(*!
<summary>Places the cursor before the first source entry.</summary>
<description>
The next MoveNext starts at zero. Does not modify the source or release payload; reading Current now yields an
empty descriptor. Descendants cannot override this cursor operation; advancement, reset and borrowed current
views use the same cursor state.
</description>
*)
{attribute "object_name" := "Reset"}
METHOD FINAL Reset
_CurrentIndex := -1;
END_METHOD

(*!
<summary>Reports the size of this function-block instance.</summary>
<description>
Measured in bytes; includes inline storage but excludes separately allocated buffers, payload and enumerators.
</description>
*)
{attribute 'monitoring' := 'call'}
PROPERTY SelfSize : ULINT
GET
SelfSize := XSIZEOF(THIS^);
END_GET
END_PROPERTY

(*!
<summary>Requires the configured source before traversal or current-value access.</summary>
<description>
A missing mandatory source is configuration failure, not an empty collection. Raises a framework diagnostic
outside lifecycle methods and before mutation; it does not validate arbitrary pointer lifetime.
</description>
*)
METHOD PRIVATE requireSource
IF _Queue = 0 THEN
	TOF_Core.Exceptions.ThrowDataMemberNotSpecified(
		sourceNamespaceName := NamespaceName,
		sourceClassName := ClassName,
		sourcePOUName := __POUNAME(),
		sourcePosition := __POSITION(),
		dataMemberName := 'queue'
	);
END_IF
END_METHOD

END_FUNCTION_BLOCK

// ---- Stack/Stack.TcPOU
(*
SPDX-FileCopyrightText: © 2026 Oleksandr Tiutyk <trofimich@gmail.com>
SPDX-License-Identifier: MIT
License: https://opensource.org/license/mit
*)

(*!
<summary>Stores generic values for last-in, first-out processing.</summary>
<description>
CreateEnumerator allocates an independent cursor owned by its caller. The collection must remain alive while
that cursor is used. Successful insertion transfers disposal responsibility for owned payload; borrowed
payload must remain alive while stored. The caller-side descriptor copy is not reset and must not be released
again after transfer. Independent owning aliases and overlapping owned allocations are unsupported. Peek and
GetByIndex borrow entries. RemoveLast releases the top without shifting remaining entries. Indices and
enumeration run from top to bottom. Static capacity defaults to ten; zero selects dynamic storage. Validators
are borrowed for the collection lifetime. ContainsGeneric defaults to releasing its query. Growth checks
allocation arithmetic and invokes the terminal mechanism on null NEW before replacing the old buffer. No
locking or mutation-version checks are implemented. Generic lookup with requested query release also attempts
cleanup on lookup failure before propagating the captured exception; terminal OOM takes precedence.
Instances cannot be assigned by value: copying backing pointers or disposal responsibility would create
unsafe aliases. Interface references still borrow this instance; copying an interface does not clone storage.
</description>
*)

{attribute 'no_explicit_call' := 'do not call this function block directly'}
FUNCTION_BLOCK FINAL Stack 
VAR_GENERIC CONSTANT
	//!<summary>Inline descriptor capacity; zero selects dynamic backing storage.</summary>
	{attribute 'hide'} 
	_StaticCapacity : TOF_Core.DINT_LENGTH := 10;
END_VAR
EXTENDS TOF_Core.Object IMPLEMENTS IStack
VAR_INPUT
	//! <summary>Number of slots added when dynamic storage is full; must be positive when growth is required.</summary>
	DefaultDynamicAllocationElementCount : BYTE := 10;	
END_VAR
VAR_STAT
	//! <summary>Class name shared by all instances of this function block.</summary>
	{attribute 'hide'} 
	_ClassName : STRING := __POUNAME();
END_VAR
VAR	
	{attribute 'hide'} 
	_ValueValidator : TOF_Core.IGenericValueValidator;

	{attribute 'hide'} 
	_Array : POINTER TO TOF_Core.GENERIC_VALUE;
	{attribute 'hide'} 
	_StaticArray : ARRAY [0.._StaticCapacity - 1] OF TOF_Core.GENERIC_VALUE;
	
	{attribute 'hide'} 
	_DynamicCapacity : TOF_Core.DINT_LENGTH;
	{attribute 'hide'} 
	_Length : TOF_Core.DINT_LENGTH;
END_VAR

(*!
<summary>Expands the dynamic descriptor buffer.</summary>
<description>
Static instances return without allocation. A positive increment must fit DINT capacity and the UDINT
allocation-byte limit; invalid ranges raise ArgumentOutOfRangeException before storage changes. A null
allocation invokes the terminal allocation-failure mechanism before copying or deleting the old buffer.
Existing descriptors are moved without cloning payload; incoming ownership is not accepted by this helper.
</description>
*)
METHOD PROTECTED FINAL AllocateMemory 
VAR_INPUT
	elementCount : TOF_Core.DINT_LENGTH;
END_VAR
VAR CONSTANT
	//!<summary>Bytes per descriptor slot used to bound and size the dynamic backing allocation.</summary>
	ENTRY_ALLOCATION_SIZE : ULINT := XSIZEOF(TOF_Core.GENERIC_VALUE);
END_VAR
VAR
	newMemory : POINTER TO TOF_Core.GENERIC_VALUE;
	newCapacity : ULINT;

END_VAR
IF NOT Dynamic THEN
	RETURN;
END_IF

IF elementCount <= TOF_Core.SignedInt32.ZERO THEN
	TOF_Core.Exceptions.ThrowArgumentOutOfRange(
		sourceNamespaceName := NamespaceName,
		sourceClassName := ClassName,
		sourcePOUName := __POUNAME(),
		sourcePosition := __POSITION(),
		argumentName := 'elementCount',
		argumentValue := elementCount
	);
END_IF

newCapacity := TO_ULINT(_DynamicCapacity) + TO_ULINT(elementCount);

IF newCapacity > TO_ULINT(TOF_Core.SignedInt32.MAX_VALUE)
	OR_ELSE newCapacity > TO_ULINT(TOF_Core.UnsignedInt32.MAX_VALUE) / ENTRY_ALLOCATION_SIZE
THEN
	TOF_Core.Exceptions.ThrowArgumentOutOfRange(
		sourceNamespaceName := NamespaceName,
		sourceClassName := ClassName,
		sourcePOUName := __POUNAME(),
		sourcePosition := __POSITION(),
		argumentName := 'capacity',
		argumentValue := newCapacity
	);
END_IF

newMemory := __NEW(BYTE, TO_UDINT(ENTRY_ALLOCATION_SIZE * newCapacity));

IF newMemory = 0 THEN
	TOF_Core.DynamicMemoryManager.RaiseAllocationFailure();
END_IF

IF _Length > TOF_Core.SignedInt32.ZERO THEN
	Tc2_System.MEMCPY(destAddr := newMemory, srcAddr := _Array, n := TO_UDINT(ENTRY_ALLOCATION_SIZE * TO_ULINT(_Length)));
END_IF

IF _Array <> 0 THEN
	__DELETE(_Array);
END_IF

_DynamicCapacity := TO_DINT(newCapacity);
_Array := newMemory;
END_METHOD

(*!
<summary>Reports the currently allocated number of slots.</summary>
<description>
Units are stack entries. Static capacity is fixed; dynamic capacity can change on growth or clearing. This is
not a guarantee that the next allocation succeeds.
</description>
*)
{attribute 'monitoring' := 'call'}
PROPERTY FINAL Capacity : TOF_Core.DINT_LENGTH
GET
Capacity := SEL(_StaticCapacity = TOF_Core.SignedInt32.ZERO, _StaticCapacity, _DynamicCapacity);
END_GET
END_PROPERTY

(*!
<summary>Borrows the concrete collection class name without transferring storage ownership.</summary>
*)
{attribute 'monitoring' := 'call'}
PROPERTY ClassName : REFERENCE TO STRING
GET
ClassName REF= _ClassName;
END_GET
END_PROPERTY

(*!
<summary>Removes all entries and releases dynamic backing storage.</summary>
<description>
Owned payload is released best effort through GENERIC_VALUE.Release; borrowed storage is not freed. Static
capacity and the borrowed validator are retained. Dynamic capacity becomes zero. Returns this collection and
invalidates positions and views. Cleanup callbacks must not reenter mutation.
</description>
*)
METHOD Clear : IStack
VAR
	i : DINT;
END_VAR
Clear := THIS^;

FOR i := 0 TO _Length - 1 DO
	_Array[i].Release();
END_FOR

_Length := 0;
_DynamicCapacity := 0;

IF _Array <> 0 AND_THEN Dynamic THEN
	__DELETE(_Array);	
END_IF
END_METHOD

(*!
<summary>Searches for a value using default generic equality.</summary>
<description>
Borrows the ANY argument during a linear search without cloning or releasing it. isObject = TRUE means a live
Object FB instance, not a pointer or interface variable. Equality exceptions propagate; callbacks that mutate
the collection can invalidate traversal.
</description>
*)
METHOD Contains : BOOL
VAR_INPUT
	value : ANY;
	isObject : BOOL := FALSE;
END_VAR
VAR
	genericValue : TOF_Core.GENERIC_VALUE;
	i : TOF_Core.DINT_INDEX;
END_VAR

genericValue := TOF_Core.GenericValueFactory.FromAnyType(
		value := value,
		isObject := isObject,
		memoryManagementBehavior := TOF_Core.GENERIC_MEMORY_MANAGEMENT_BEHAVIOR.STORE_ORIGINAL_REFERENCE_AND_NOT_OWNS_MEMORY
	);

FOR i := 0 TO _Length - 1 DO
	IF _Array[i].Equals(otherValue := genericValue) THEN
		Contains := TRUE;
		RETURN;
	END_IF
END_FOR
END_METHOD

(*!
<summary>Searches for an equal generic value and optionally releases the query.</summary>
<description>
Uses GENERIC_VALUE.Equals in a linear search. releaseValue defaults to TRUE: after a completed search, Release
is called on the local query copy, including on a miss. Caller-side aliases are not reset. The query must not
own storage retained by the collection. Requested release is attempted after both successful lookup and lookup
failure. Before cleanup, the original framework exception is retained and a borrowed static system exception
is cloned to preserve its code, catch point and timestamps across cleanup callbacks. The captured exception is
then propagated through ExceptionManager.Throw in the current cyclic task; native errors use the framework
SystemException representation. If capturing the system exception fails with terminal OOM, query cleanup is
still attempted and terminal OOM takes precedence. Terminal allocation state is never cleared. Release is best
effort and does not prove successful deallocation. Cleanup callbacks must not reenter collection mutation.
</description>
*)
METHOD ContainsGeneric : BOOL
VAR_INPUT
	value : TOF_Core.GENERIC_VALUE;
	releaseValue : BOOL := TRUE;
END_VAR
VAR
	exceptionCode : __SYSTEM.ExceptionCode;
	caughtException : TOF_Core.IException;

	i : DINT;
END_VAR
__TRY
	FOR i := 0 TO _Length - 1 DO
		IF _Array[i].Equals(otherValue := value) THEN
			ContainsGeneric := TRUE;
			EXIT;
		END_IF
	END_FOR
__CATCH(exceptionCode)
	caughtException := TOF_Core.ExceptionManager.GetLastException(
		exceptionCode := exceptionCode,
		catchPointNamespaceName := NamespaceName,
		catchPointPOUName := __POUNAME(),
		catchPointPosition := __POSITION()
	);
__ENDTRY

IF releaseValue THEN
	IF caughtException <> 0 AND_THEN NOT caughtException.IsDynamicInstance THEN
		__TRY
			TOF_Core.DynamicMemoryManager.RaiseIfAllocationFailed();
			__QUERYINTERFACE(caughtException.Clone(), caughtException);
		__CATCH(exceptionCode)
			value.Release();

			TOF_Core.ExceptionManager.ReThrowLastException(
				exceptionCode := exceptionCode,
				catchPointNamespaceName := NamespaceName,
				catchPointPOUName := __POUNAME(),
				catchPointPosition := __POSITION()
			);
		__ENDTRY
	END_IF

	value.Release();
END_IF

IF caughtException <> 0 THEN
	TOF_Core.ExceptionManager.Throw(exception := caughtException);
END_IF
END_METHOD

(*!
<summary>Creates an independent enumerator owned by the caller.</summary>
<description>
The caller must explicitly release the enumerator and keep this collection alive while using it. Allocation
failure invokes DynamicMemoryManager.RaiseAllocationFailure without a heap exception; it is terminal and is
not returned as a recoverable null result.
</description>
*)
METHOD CreateEnumerator : TOF_Core.IEnumerator
VAR
	enumerator : POINTER TO StackEnumerator;
END_VAR
enumerator := __NEW(StackEnumerator(stack := THIS^));

IF enumerator = 0 THEN
	TOF_Core.DynamicMemoryManager.RaiseAllocationFailure();
END_IF

CreateEnumerator := enumerator^;
END_METHOD

(*!
<summary>Reports whether storage can grow dynamically.</summary>
<description>
Static capacity zero selects dynamic storage. Dynamic collections can still fail to allocate.
</description>
*)
{attribute 'monitoring' := 'call'}
PROPERTY FINAL Dynamic : BOOL
GET
Dynamic := _StaticCapacity = TOF_Core.SignedInt32.ZERO;
END_GET
END_PROPERTY

(*!
<summary>Reports whether the collection has no entries.</summary>
<description>
Reflects Length; not a check of payload lifetime or memory health.
</description>
*)
{attribute 'monitoring' := 'call'}
PROPERTY FINAL Empty : BOOL
GET
Empty := _Length <= TOF_Core.SignedInt32.ZERO;
END_GET
END_PROPERTY

(*!
<summary>Releases owned payload and backing storage during destruction.</summary>
<description>
Calls Clear; lifecycle methods and payload cleanup callbacks must not raise exceptions or reenter mutation.
Payload release is best effort, not proof of successful destruction. No separate copy-code ownership handoff
is implemented.
</description>
*)

METHOD FB_exit : BOOL
VAR_INPUT
	bInCopyCode : BOOL; 
END_VAR
Clear();
END_METHOD

(*!
<summary>Binds the optional validator and inline storage during initialization.</summary>
<description>
The validator is borrowed and must remain alive while used; it is not invoked here. Static storage is bound
without allocation. Lifecycle methods must not raise exceptions. No explicit online-change relocation repair
is implemented.
</description>
*)
METHOD FB_init : BOOL
VAR_INPUT
	bInitRetains : BOOL; // TRUE: the retain variables are initialized (reset warm / reset cold)
	bInCopyCode : BOOL; // TRUE: the instance will be copied to the copy code afterward (online change)
	valueValidator : TOF_Core.IGenericValueValidator;
END_VAR
_ValueValidator := valueValidator;

IF NOT Dynamic THEN
	_Array := ADR(_StaticArray); 
END_IF
END_METHOD

(*!
<summary>Reports whether fixed-capacity storage has no free slot.</summary>
<description>
Dynamic collections report FALSE even when Length equals Capacity. This does not guarantee available heap
memory.
</description>
*)
{attribute 'monitoring' := 'call'}
PROPERTY FINAL Full : BOOL
GET
Full := _StaticCapacity <> TOF_Core.SignedInt32.ZERO AND_THEN _Length >= _StaticCapacity;
END_GET
END_PROPERTY

(*!
<summary>Borrows the descriptor at a zero-based stack position.</summary>
<description>
Position zero is the top; increasing indices move toward the bottom. An out-of-range index raises an
exception. Returned descriptors and payload are borrowed, not clones. Do not modify descriptor metadata or
release payload through this view, even when IsMemoryOwner is TRUE. Keep the source and borrowed storage
alive; mutation or destruction can invalidate the view.
</description>
*)
METHOD GetByIndex : REFERENCE TO TOF_Core.GENERIC_VALUE
VAR_INPUT
	index : TOF_Core.DINT_INDEX;
END_VAR
IF index < TOF_Core.SignedInt32.ZERO OR_ELSE index >= _Length THEN
	TOF_Core.Exceptions.ThrowArgumentOutOfRange(
		sourceNamespaceName := NamespaceName,
		sourceClassName := ClassName,
		sourcePOUName := __POUNAME(),
		sourcePosition := __POSITION(),
		argumentName := 'index',
		argumentValue := index
	);
END_IF

GetByIndex REF= _Array[_Length - 1 - index];
END_METHOD

(*!
<summary>Reports the number of stored entries.</summary>
<description>
Units are stack entries. Existing positions range from zero through Length minus one.
</description>
*)
{attribute 'monitoring' := 'call'}
PROPERTY FINAL Length : TOF_Core.DINT_LENGTH
GET
Length := _Length;
END_GET
END_PROPERTY

(*!
<summary>Provides the library namespace for diagnostics.</summary>
<description>
Borrowed read-only reference to compiler-initialized metadata; no ownership transfer.
</description>
*)
{attribute 'monitoring' := 'call'}
PROPERTY NamespaceName : REFERENCE TO STRING
GET
NamespaceName REF= CurrentNamespace.Name;
END_GET
END_PROPERTY

(*!
<summary>Borrows the LIFO top without removing it.</summary>
<description>
An empty stack raises CollectionEmptyException. Returned descriptors and payload are borrowed, not clones. Do
not modify descriptor metadata or release payload through this view, even when IsMemoryOwner is TRUE. Keep the
source and borrowed storage alive; mutation or destruction can invalidate the view.
</description>
*)
METHOD Peek : REFERENCE TO TOF_Core.GENERIC_VALUE
IF _Length <= TOF_Core.SignedInt32.ZERO THEN
	TOF_Core.Exceptions.ThrowCollectionEmpty(
		sourceNamespaceName := NamespaceName,
		sourceClassName := ClassName,
		sourcePOUName := __POUNAME(),
		sourcePosition := __POSITION(),
		collectionName := GetName()
	);
END_IF

Peek REF= _Array[_Length - 1];
END_METHOD

(*!
<summary>Copies a value and appends it to the stack top.</summary>
<description>
Borrows the original during the call. isObject = TRUE requires a live Object FB instance implementing
ICloneable; other data is copied as bytes without recursively cloning references. A prepared copy is released
if insertion fails before acceptance; exceptions propagate. Engine-managed exception objects are unsupported.
The original failure is captured before cleanup so nested cleanup handling cannot replace its payload.
A static native wrapper is cloned before cleanup; failure to capture still attempts prepared-copy disposal.
Terminal allocation failure takes precedence and no exception clone is allocated after its latch is set.
</description>
*)
METHOD PushCopy : IStack
VAR_INPUT
	value : ANY;
	isObject : BOOL := FALSE;
END_VAR
VAR
	exceptionCode : __SYSTEM.ExceptionCode;
	caughtException : TOF_Core.IException;
	genericValue : TOF_Core.GENERIC_VALUE;
END_VAR

genericValue := TOF_Core.GenericValueFactory.FromAnyType(
		value := value,
		isObject := isObject,
		memoryManagementBehavior := TOF_Core.GENERIC_MEMORY_MANAGEMENT_BEHAVIOR.CLONE_ORIGINAL_VALUE_AND_OWNS_MEMORY
	);

__TRY
	PushCopy := PushGeneric(value := genericValue);
__CATCH(exceptionCode)
	caughtException := TOF_Core.ExceptionManager.GetLastException(
		exceptionCode := exceptionCode,
		catchPointNamespaceName := NamespaceName,
		catchPointPOUName := __POUNAME(),
		catchPointPosition := __POSITION()
	);
__ENDTRY

IF caughtException <> 0 THEN
	__TRY
		TOF_Core.DynamicMemoryManager.RaiseIfAllocationFailed();

		IF NOT caughtException.IsDynamicInstance THEN
			__QUERYINTERFACE(caughtException.Clone(), caughtException);
		END_IF
	__CATCH(exceptionCode)
		genericValue.Release();

		TOF_Core.ExceptionManager.ReThrowLastException(
			exceptionCode := exceptionCode,
			catchPointNamespaceName := NamespaceName,
			catchPointPOUName := __POUNAME(),
			catchPointPosition := __POSITION()
		);
	__ENDTRY

	genericValue.Release();

	TOF_Core.ExceptionManager.Throw(exception := caughtException);
END_IF
END_METHOD

(*!
<summary>Pushes a descriptor onto the stack top.</summary>
<description>
Successful insertion transfers disposal responsibility for owned payload; borrowed payload must remain alive
while stored. The caller-side descriptor copy is not reset and must not be released again after transfer.
Independent owning aliases and overlapping owned allocations are unsupported. Full static storage raises an
exception. A configured validator is invoked once before any capacity growth or ownership acceptance.
Validation failure leaves the buffer, Length and incoming ownership unchanged; its exception propagates.
Validator callbacks must not mutate this collection.
</description>
*)
METHOD PushGeneric : IStack
VAR_INPUT
	value : TOF_Core.GENERIC_VALUE;
END_VAR
IF _ValueValidator <> 0 THEN
	_ValueValidator.Validate(validatedObjectName := GetName(), valueToValidate := value);
END_IF

IF _Length >= Capacity THEN
	IF Dynamic THEN
		AllocateMemory(elementCount := DefaultDynamicAllocationElementCount);
	ELSE
		TOF_Core.Exceptions.ThrowStaticCollectionFull(
			sourceNamespaceName := NamespaceName,
			sourceClassName := ClassName,
			sourcePOUName := __POUNAME(),
			sourcePosition := __POSITION(),
			collectionName := GetName(),
			capacity := TO_UDINT(Capacity)
		);
	END_IF
END_IF

PushGeneric := THIS^;

_Array[_Length] := value;
_Length := _Length + 1;
END_METHOD

(*!
<summary>Removes and releases the LIFO top.</summary>
<description>
An empty stack raises CollectionEmptyException. Owned top storage is released best effort, not returned to the
caller. Remaining descriptors are not moved; removal takes constant time apart from payload cleanup. Returns
this stack; positions and views may change. Cleanup callbacks must not reenter mutation.
</description>
*)
METHOD RemoveLast : IStack
IF _Length <= TOF_Core.SignedInt32.ZERO THEN
	TOF_Core.Exceptions.ThrowCollectionEmpty(
		sourceNamespaceName := NamespaceName,
		sourceClassName := ClassName,
		sourcePOUName := __POUNAME(),
		sourcePosition := __POSITION(),
		collectionName := GetName()
	);
END_IF

_Length := _Length - 1;
_Array[_Length].Release();

RemoveLast := THIS^;
END_METHOD

(*!
<summary>Reports the size of this function-block instance.</summary>
<description>
Measured in bytes; includes inline storage but excludes separately allocated buffers, payload and enumerators.
</description>
*)
{attribute 'monitoring' := 'call'}
PROPERTY SelfSize : ULINT
GET
SelfSize := XSIZEOF(THIS^);
END_GET
END_PROPERTY

(*!
<summary>Exposes the configured value validator.</summary>
<description>
Borrowed optional reference fixed at initialization. Zero means no validator. The collection does not own or
release it.
</description>
*)
{attribute 'monitoring' := 'call'}
PROPERTY FINAL ValueValidator : TOF_Core.IGenericValueValidator
GET
ValueValidator := _ValueValidator;
END_GET
END_PROPERTY

END_FUNCTION_BLOCK

// ---- Stack/StackEnumerator.TcPOU
(*
SPDX-FileCopyrightText: © 2026 Oleksandr Tiutyk <trofimich@gmail.com>
SPDX-License-Identifier: MIT
License: https://opensource.org/license/mit
*)

(*!
<summary>Enumerates a borrowed stack using an independent cursor.</summary>
<description>
The source must be non-null, outlive the cursor and remain structurally unchanged during traversal. The caller
explicitly releases a dynamically created cursor. Current is borrowed read-only data, never an ownership
transfer. Traverses from top to bottom. Supports both fixed-capacity and dynamic stacks. MoveNext stops
advancing at the end position of an unchanged source; repeated exhausted calls return FALSE until Reset.
A null constructor source is diagnosed by traversal/current access, never by FB_init.
</description>
*)

{attribute 'no_explicit_call' := 'do not call this function block directly'}
{attribute 'enable_dynamic_creation'}
FUNCTION_BLOCK StackEnumerator EXTENDS TOF_Core.Object IMPLEMENTS TOF_Core.IEnumerator
VAR_STAT
	//! <summary>Class name shared by all instances of this function block.</summary>
	{attribute 'hide'} 
	_ClassName : STRING := __POUNAME();
END_VAR
VAR
	{attribute 'hide'} 
	_Stack : IReadOnlyStack;
	{attribute 'hide'} 
	//!<summary>Top-relative position; minus one represents the cursor before the first entry.</summary>
	_CurrentIndex : DINT := -1;
	
	{attribute 'hide'} 
	_GenericValue : TOF_Core.GENERIC_VALUE;
END_VAR

(*!
<summary>Borrows the concrete cursor class name without transferring storage ownership.</summary>
*)
{attribute 'monitoring' := 'call'}
PROPERTY ClassName : REFERENCE TO STRING
GET
ClassName REF= _ClassName;
END_GET
END_PROPERTY

(*!
<summary>Exposes a read-only borrowed view of the current entry.</summary>
<description>
Reading Current before the first successful MoveNext, after Reset or after exhaustion yields an empty
descriptor. Otherwise payload is borrowed, with no disposal rights. Do not modify or release the descriptor.
The view may change on subsequent property access, cursor movement or source mutation.
Missing source raises DataMemberNotSpecifiedException before source access or cursor advancement.
</description>
*)
{attribute 'monitoring' := 'call'}
PROPERTY FINAL Current : REFERENCE TO TOF_Core.GENERIC_VALUE
GET
requireSource();

IF _CurrentIndex >= TOF_Core.SignedInt32.ZERO AND_THEN _CurrentIndex < _Stack.Length THEN
	_GenericValue := _Stack.GetByIndex(index := _CurrentIndex); 
ELSE
	_GenericValue.Reset();	
END_IF 

Current REF= _GenericValue;
END_GET
END_PROPERTY

(*!
<summary>Binds the borrowed source for enumeration.</summary>
<description>
The source must be non-null and outlive the cursor. Only the reference is assigned; no allocation, callbacks
or throwing validation are performed. A null source remains invalid configuration and is reported by
MoveNext or current-value access without throwing from initialization.
</description>
*)
METHOD FB_init : BOOL
VAR_INPUT
	bInitRetains : BOOL; // TRUE: the retain variables are initialized (reset warm / reset cold)
	bInCopyCode : BOOL;  // TRUE: the instance will be copied to the copy code afterward (online change)
	stack : IReadOnlyStack;
END_VAR
_Stack := stack;
END_METHOD

(*!
<summary>Advances the cursor to the next source position.</summary>
<description>
The source must be live, non-null and structurally unchanged during traversal. TRUE identifies a current
entry. The index advances only while below source Length and stops at the end position. Repeated exhausted
calls return FALSE without incrementing the index; reading Current yields an empty descriptor. Reset allows
traversal from the beginning again. No snapshot or mutation detection is provided. Descendants cannot override
this cursor operation; advancement, reset and borrowed current views use the same cursor state.
Missing source raises DataMemberNotSpecifiedException before source access or cursor advancement.
</description>
*)
{attribute "object_name" := "MoveNext"}
METHOD FINAL MoveNext : BOOL
requireSource();

IF _CurrentIndex < _Stack.Length THEN
	_CurrentIndex := _CurrentIndex + 1;
END_IF

MoveNext := _CurrentIndex < _Stack.Length;
END_METHOD

(*!
<summary>Provides the library namespace for diagnostics.</summary>
<description>
Borrowed read-only reference to compiler-initialized metadata; no ownership transfer.
</description>
*)
{attribute 'monitoring' := 'call'}
PROPERTY NamespaceName : REFERENCE TO STRING
GET
NamespaceName REF= CurrentNamespace.Name;
END_GET
END_PROPERTY

(*!
<summary>Places the cursor before the first source entry.</summary>
<description>
The next MoveNext starts at zero. Does not modify the source or release payload; reading Current now yields an
empty descriptor. Descendants cannot override this cursor operation; advancement, reset and borrowed current
views use the same cursor state.
</description>
*)
{attribute "object_name" := "Reset"}
METHOD FINAL Reset
_CurrentIndex := -1;
END_METHOD

(*!
<summary>Reports the size of this function-block instance.</summary>
<description>
Measured in bytes; includes inline storage but excludes separately allocated buffers, payload and enumerators.
</description>
*)
{attribute 'monitoring' := 'call'}
PROPERTY SelfSize : ULINT
GET
SelfSize := XSIZEOF(THIS^);
END_GET
END_PROPERTY

(*!
<summary>Requires the configured source before traversal or current-value access.</summary>
<description>
A missing mandatory source is configuration failure, not an empty collection. Raises a framework diagnostic
outside lifecycle methods and before mutation; it does not validate arbitrary pointer lifetime.
</description>
*)
METHOD PRIVATE requireSource
IF _Stack = 0 THEN
	TOF_Core.Exceptions.ThrowDataMemberNotSpecified(
		sourceNamespaceName := NamespaceName,
		sourceClassName := ClassName,
		sourcePOUName := __POUNAME(),
		sourcePosition := __POSITION(),
		dataMemberName := 'stack'
	);
END_IF
END_METHOD

END_FUNCTION_BLOCK

// ---- UniqueDataSet/UniqueDataSet.TcPOU
(*
SPDX-FileCopyrightText: © 2026 Oleksandr Tiutyk <trofimich@gmail.com>
SPDX-License-Identifier: MIT
License: https://opensource.org/license/mit
*)

(*!
<summary>Stores unique generic values with fixed or dynamic capacity.</summary>
<description>
CreateEnumerator allocates an independent cursor owned by its caller. The collection must remain alive while
that cursor is used. SetGeneric replaces a matching entry with the incoming descriptor. SetGeneric preserves
disposal responsibility when the same allocation is reused; transferred caller-side owning aliases must not be
released again. Lookup uses GENERIC_VALUE equality/hashing or the borrowed valueEqualityComparer supplied once
through FB_init. Pass zero explicitly to use default value equality and hashing. Empty values are supported
unless rejected by a validator. Raw queries create borrowed descriptors with an explicit object flag. Entries
and enumeration have no guaranteed order; positions are storage slots, not sorted ranks. Do not modify stored
descriptors through returned references. Try lookup/removal operations contain exceptions without rolling back
partial effects. Generic query arguments are borrowed by default. Explicitly requested release in Try
operations is attempted even after lookup failure; caller-side owning aliases are not reset. Borrowed
elements, including OBJECT instances, remain caller-owned and must stay alive while stored. Do not delete
owned payload through external aliases. Keep equality/hash-relevant data and comparer configuration stable:
remove before changing them, then insert again. Fields unrelated to active equality/hash may change. Callbacks
must not mutate elements or reenter collection mutation; explicit query release must not dispose of retained
storage. Default OBJECT equality/hashing uses Object.Equals/GetHashCode; Clone has its own identity. Discard
and populate the index again after equality-relevant address relocation before further lookup. Static index
storage adds 12 bytes per capacity slot and three pointers plus the comparer reference. Dynamic entries and
the 12-byte-per-slot index share one allocation; growth temporarily retains both old and new allocations.
Expected bucket lookup is constant time plus hashing/equality costs, worst case linear; compaction and
rebuilding after removal are linear in capacity and Length. The validator is borrowed for the collection
lifetime. No internal locking is implemented. Concurrent access involving mutation requires caller
coordination; this implementation does not provide a concurrent-container guarantee. Generic lookup with
requested query release also attempts cleanup on lookup failure before propagating the captured exception;
terminal OOM takes precedence.
Instances cannot be assigned by value: copying backing pointers or disposal responsibility would create
unsafe aliases. Interface references still borrow this instance; copying an interface does not clone storage.
</description>
*)

{attribute 'no_explicit_call' := 'do not call this function block directly'}
FUNCTION_BLOCK UniqueDataSet
VAR_GENERIC CONSTANT
	{attribute 'hide'}
	//! <summary>Inline capacity; zero selects dynamic backing storage.</summary>
	_StaticCapacity : TOF_Core.DINT_LENGTH := 0;
END_VAR
EXTENDS TOF_Core.Object IMPLEMENTS IUniqueDataSet
VAR_INPUT
	//! <summary>Number of slots added when dynamic storage is full; must be positive when growth is required.</summary>
	DefaultDynamicAllocationElementCount : BYTE := 10;
END_VAR
VAR_STAT
	//! <summary>Class name shared by all instances of this function block.</summary>
	{attribute 'hide'}
	_ClassName : STRING := __POUNAME();
END_VAR
VAR
	{attribute 'hide'}
	_ValueValidator : TOF_Core.IGenericValueValidator;
	{attribute 'hide'}
	_ValueEqualityComparer : TOF_Core.IEqualityComparer;

	{attribute 'hide'}
	_Array : POINTER TO TOF_Core.GENERIC_VALUE;
	{attribute 'hide'}
	_StaticArray : ARRAY [0.._StaticCapacity - 1] OF TOF_Core.GENERIC_VALUE;

	{attribute 'hide'}
	_Hashes : POINTER TO UDINT;
	{attribute 'hide'}
	_Buckets : POINTER TO DINT;
	{attribute 'hide'}
	_NextIndices : POINTER TO DINT;

	{attribute 'hide'}
	_StaticHashes : ARRAY [0.._StaticCapacity - 1] OF UDINT;
	{attribute 'hide'}
	_StaticBuckets : ARRAY [0.._StaticCapacity - 1] OF DINT;
	{attribute 'hide'}
	_StaticNextIndices : ARRAY [0.._StaticCapacity - 1] OF DINT;

	{attribute 'hide'}
	_DynamicCapacity : TOF_Core.DINT_LENGTH;
	{attribute 'hide'}
	_Length : TOF_Core.DINT_LENGTH;
END_VAR

(*!
<summary>Grows the combined entry and hash-index buffer before accepting incoming ownership.</summary>
<description>
Static collections return without allocation. A positive increment must fit DINT capacity and the UDINT
allocation-byte limit, including 12 index bytes per slot. One allocation contains entries, cached hashes,
bucket heads and links. Allocation failure preserves the old buffer, index, capacity and payload ownership and
sets terminal allocation state. Existing descriptors and hashes are copied; rebuilding links invokes no
equality/hash callbacks. Descendants cannot override this storage operation; capacity, indexing and disposal
remain governed by this collection implementation.
</description>
*)
METHOD PROTECTED FINAL AllocateMemory
VAR_INPUT
	elementCount : TOF_Core.DINT_LENGTH;
END_VAR
VAR CONSTANT
	//! <summary>Bytes per capacity slot, including descriptor storage and any hash-index arrays.</summary>
	ENTRY_ALLOCATION_SIZE : ULINT := XSIZEOF(TOF_Core.GENERIC_VALUE) + XSIZEOF(UDINT) + 2 * XSIZEOF(DINT);
END_VAR
VAR
	newMemory : POINTER TO BYTE;
	newHashes : POINTER TO UDINT;
	newCapacity : ULINT;

END_VAR
IF NOT Dynamic THEN
	RETURN;
END_IF

IF elementCount <= TOF_Core.SignedInt32.ZERO THEN
	TOF_Core.Exceptions.ThrowArgumentOutOfRange(
		sourceNamespaceName := NamespaceName,
		sourceClassName := ClassName,
		sourcePOUName := __POUNAME(),
		sourcePosition := __POSITION(),
		argumentName := 'elementCount',
		argumentValue := elementCount
	);
END_IF

newCapacity := TO_ULINT(_DynamicCapacity) + TO_ULINT(elementCount);

IF newCapacity > TO_ULINT(TOF_Core.SignedInt32.MAX_VALUE)
	OR_ELSE newCapacity > TO_ULINT(TOF_Core.UnsignedInt32.MAX_VALUE) / ENTRY_ALLOCATION_SIZE
THEN
	TOF_Core.Exceptions.ThrowArgumentOutOfRange(
		sourceNamespaceName := NamespaceName,
		sourceClassName := ClassName,
		sourcePOUName := __POUNAME(),
		sourcePosition := __POSITION(),
		argumentName := 'capacity',
		argumentValue := newCapacity
	);
END_IF

newMemory := __NEW(BYTE, TO_UDINT(ENTRY_ALLOCATION_SIZE * newCapacity));

IF newMemory = 0 THEN
	TOF_Core.DynamicMemoryManager.RaiseAllocationFailure();
END_IF

newHashes := newMemory + TO_UDINT(XSIZEOF(TOF_Core.GENERIC_VALUE) * newCapacity);

IF _Length > TOF_Core.SignedInt32.ZERO THEN
	Tc2_System.MEMCPY(
		destAddr := newMemory,
		srcAddr := _Array,
		n := TO_UDINT(XSIZEOF(TOF_Core.GENERIC_VALUE) * TO_ULINT(_Length))
	);
	Tc2_System.MEMCPY(destAddr := newHashes, srcAddr := _Hashes, n := TO_UDINT(XSIZEOF(UDINT) * TO_ULINT(_Length)));
END_IF

IF _Array <> 0 THEN
	__DELETE(_Array);
END_IF

_Array := newMemory;
_Hashes := newHashes;
_Buckets := newMemory + TO_UDINT((XSIZEOF(TOF_Core.GENERIC_VALUE) + XSIZEOF(UDINT)) * newCapacity);
_NextIndices := newMemory + TO_UDINT((XSIZEOF(TOF_Core.GENERIC_VALUE) + XSIZEOF(UDINT) + XSIZEOF(DINT)) * newCapacity);
_DynamicCapacity := TO_DINT(newCapacity);

rebuildIndex();
END_METHOD

(*!
<summary>Reports the currently allocated number of slots.</summary>
<description>
Units are bytes for ByteList and entries for other collections. Static capacity is fixed; dynamic capacity can
change on growth or clearing. This is not a guarantee that the next allocation succeeds.
</description>
*)
{attribute 'monitoring' := 'call'}
PROPERTY FINAL Capacity : TOF_Core.DINT_LENGTH
GET
Capacity := SEL(_StaticCapacity = 0, _StaticCapacity, _DynamicCapacity);
END_GET
END_PROPERTY

(*!
<summary>Borrows the concrete collection class name without transferring storage ownership.</summary>
*)
{attribute 'monitoring' := 'call'}
PROPERTY ClassName : REFERENCE TO STRING
GET
ClassName REF= _ClassName;
END_GET
END_PROPERTY

(*!
<summary>Removes all entries and releases dynamic entry and index storage.</summary>
<description>
Owned payload cleanup is best effort. The collection is marked empty before disposal; cleanup callbacks must
not reenter mutation. Static capacity and the lifetime comparer/validators are retained. Dynamic capacity
becomes zero. Uses no allocation or equality/hash callbacks and leaves static buckets empty for reuse.
Descendants cannot override this storage operation; capacity, indexing and disposal remain governed by this
collection implementation.
</description>
*)
METHOD FINAL Clear : IUniqueDataSet
VAR
	index : DINT;
	entryCount : DINT;
END_VAR
Clear := THIS^;
entryCount := _Length;
_Length := 0;

FOR index := 0 TO entryCount - 1 DO
	_Array[index].Release();
END_FOR

IF Dynamic THEN
	IF _Array <> 0 THEN
		__DELETE(_Array);
	END_IF

	_Array := 0;
	_Hashes := 0;
	_Buckets := 0;
	_NextIndices := 0;
	_DynamicCapacity := 0;
ELSE
	rebuildIndex();
END_IF
END_METHOD

(*!
<summary>Reports whether a matching raw query exists.</summary>
<description>
The raw ANY argument is borrowed without cloning or ownership transfer. isObject = TRUE requires a live Object
function-block instance, not a pointer or interface variable. FALSE uses ordinary runtime type mapping. The
caller keeps the query storage alive for the call. Descendants cannot override this storage operation;
capacity, indexing and disposal remain governed by this collection implementation.
</description>
*)
//!<param name="isObject">Explicitly interprets the raw argument as a live Object instance.</param>
METHOD FINAL Contains : BOOL
VAR_INPUT
	value : ANY;
	isObject : BOOL := FALSE;
END_VAR
VAR
	genericValue : TOF_Core.GENERIC_VALUE;
END_VAR

genericValue := TOF_Core.GenericValueFactory.FromAnyType(
		value := value,
		isObject := isObject,
		memoryManagementBehavior := TOF_Core.GENERIC_MEMORY_MANAGEMENT_BEHAVIOR.STORE_ORIGINAL_REFERENCE_AND_NOT_OWNS_MEMORY
	);

Contains := FindIndex(value := genericValue);
END_METHOD

(*!
<summary>Reports whether a matching entry exists for a borrowed generic query.</summary>
<description>
The query is borrowed by default. Explicit release requests disposal of owned query storage after lookup
completes, including a missing result. Requested release is attempted after both successful lookup and lookup
failure. Before cleanup, the original framework exception is retained and a borrowed static system exception
is cloned to preserve its code, catch point and timestamps across cleanup callbacks. The captured exception is
then propagated through ExceptionManager.Throw in the current cyclic task; native errors use the framework
SystemException representation. If capturing the system exception fails with terminal OOM, query cleanup is
still attempted and terminal OOM takes precedence. Terminal allocation state is never cleared. Release is best
effort and does not prove successful deallocation. Cleanup callbacks must not reenter collection mutation.
Release resets only the local descriptor copy; the caller must have disposal rights and must not reuse or
release owning aliases afterwards. Borrowed payload is not freed. Descendants cannot override this storage
operation; capacity, indexing and disposal remain governed by this collection implementation.
</description>
*)
METHOD FINAL ContainsGeneric : BOOL
VAR_INPUT
	value : TOF_Core.GENERIC_VALUE;
	releaseValue : BOOL := FALSE;
END_VAR
VAR
	exceptionCode : __SYSTEM.ExceptionCode;
	caughtException : TOF_Core.IException;
END_VAR
__TRY
	ContainsGeneric := FindIndex(value := value);
__CATCH(exceptionCode)
	caughtException := TOF_Core.ExceptionManager.GetLastException(
		exceptionCode := exceptionCode,
		catchPointNamespaceName := NamespaceName,
		catchPointPOUName := __POUNAME(),
		catchPointPosition := __POSITION()
	);
__ENDTRY

IF releaseValue THEN
	IF caughtException <> 0 AND_THEN NOT caughtException.IsDynamicInstance THEN
		__TRY
			TOF_Core.DynamicMemoryManager.RaiseIfAllocationFailed();
			__QUERYINTERFACE(caughtException.Clone(), caughtException);
		__CATCH(exceptionCode)
			value.Release();

			TOF_Core.ExceptionManager.ReThrowLastException(
				exceptionCode := exceptionCode,
				catchPointNamespaceName := NamespaceName,
				catchPointPOUName := __POUNAME(),
				catchPointPosition := __POSITION()
			);
		__ENDTRY
	END_IF

	value.Release();
END_IF

IF caughtException <> 0 THEN
	TOF_Core.ExceptionManager.Throw(exception := caughtException);
END_IF
END_METHOD

(*!
<summary>Creates an independent enumerator owned by the caller.</summary>
<description>
The caller must explicitly release the enumerator and keep this collection alive while using it. Allocation
failure invokes DynamicMemoryManager.RaiseAllocationFailure without a heap exception; it is terminal and is
not returned as a recoverable null result.
</description>
*)
METHOD CreateEnumerator : TOF_Core.IEnumerator
VAR
	enumerator : POINTER TO UniqueDataSetEnumerator;
END_VAR
enumerator := __NEW(UniqueDataSetEnumerator(uniqueSet := THIS^));

IF enumerator = 0 THEN
	TOF_Core.DynamicMemoryManager.RaiseAllocationFailure();
END_IF

CreateEnumerator := enumerator^;
END_METHOD

(*!
<summary>Reports whether storage can grow dynamically.</summary>
<description>
Static capacity zero selects dynamic storage. Dynamic collections can still fail to allocate.
</description>
*)
{attribute 'monitoring' := 'call'}
PROPERTY FINAL Dynamic : BOOL
GET
Dynamic := _StaticCapacity = 0;
END_GET
END_PROPERTY

(*!
<summary>Reports whether the collection has no entries.</summary>
<description>
Reflects Length; not a check of payload lifetime or memory health.
</description>
*)
{attribute 'monitoring' := 'call'}
PROPERTY FINAL Empty : BOOL
GET
Empty := _Length <= 0;
END_GET
END_PROPERTY

(*!
<summary>Releases collection payload and dynamic entry/index storage during destruction.</summary>
<description>
Calls the non-allocating Clear path without invoking equality/hash callbacks. Owned payload release is best
effort and cannot guarantee successful deallocation; cleanup callbacks must not throw or reenter mutation.
</description>
*)

METHOD FB_exit : BOOL
VAR_INPUT
	bInCopyCode : BOOL;
END_VAR
Clear();
END_METHOD

(*!
<summary>Binds the validator, the lifetime equality strategy and static storage.</summary>
<description>
The value comparer is borrowed for the entire collection lifetime. Supply it explicitly; zero selects
GENERIC_VALUE default equality and hashing. Keep it alive and its equality-relevant configuration stable.
There is no subsequent comparer replacement. Initialization binds existing storage without allocating or
calling validators, comparers or other throwing paths.
</description>
*)


//!<param name="valueEqualityComparer">
//! Borrowed value equality and hash strategy; pass zero explicitly for the GENERIC_VALUE defaults.
//! </param>
METHOD FB_init : BOOL
VAR_INPUT
	bInitRetains : BOOL; // TRUE: the retain variables are initialized (reset warm / reset cold)
	bInCopyCode : BOOL; // TRUE: the instance will be copied to the copy code afterward (online change)

	valueValidator : TOF_Core.IGenericValueValidator;
	valueEqualityComparer : TOF_Core.IEqualityComparer;
END_VAR
_ValueValidator := valueValidator;
_ValueEqualityComparer := valueEqualityComparer;

IF NOT Dynamic THEN
	_Array := ADR(_StaticArray);
	_Hashes := ADR(_StaticHashes);
	_Buckets := ADR(_StaticBuckets);
	_NextIndices := ADR(_StaticNextIndices);
END_IF
END_METHOD

(*!
<summary>Finds an equal value through its hash bucket.</summary>
<description>
Borrows the descriptor and payload without changing ownership. The configured equality strategy computes the
query hash once; equal hash codes are resolved with Equals. Callback exceptions propagate before mutation. On
a miss supposedIndex is the append position. hashCode is valid after a completed lookup, including a miss. No
ordering or sorted rank is provided. Bucket heads and links encode entry index plus one; zero ends a chain.
Descendants cannot override this storage operation; capacity, indexing and disposal remain governed by this
collection implementation.
</description>
*)
METHOD PROTECTED FINAL FindIndex : BOOL
VAR_INPUT
	value : TOF_Core.GENERIC_VALUE;
END_VAR
VAR_OUTPUT
	supposedIndex : DINT;
	hashCode : UDINT;
END_VAR
VAR
	entryLink : DINT;
	entryIndex : DINT;
END_VAR
FindIndex := FALSE;
supposedIndex := _Length;
hashCode := value.GetHashCode(comparer := _ValueEqualityComparer);

IF _Length = TOF_Core.SignedInt32.ZERO THEN
	RETURN;
END_IF

entryLink := _Buckets[TO_DINT(hashCode MOD TO_UDINT(Capacity))];

WHILE entryLink <> TOF_Core.SignedInt32.ZERO DO
	entryIndex := entryLink - 1;

	IF _Hashes[entryIndex] = hashCode
		AND_THEN _Array[entryIndex].Equals(otherValue := value, comparer := _ValueEqualityComparer)
	THEN
		supposedIndex := entryIndex;
		FindIndex := TRUE;
		RETURN;
	END_IF

	entryLink := _NextIndices[entryIndex];
END_WHILE
END_METHOD

(*!
<summary>Reports whether fixed-capacity storage has no free slot.</summary>
<description>
Dynamic collections report FALSE even when Length equals Capacity. This does not guarantee available heap
memory.
</description>
*)
{attribute 'monitoring' := 'call'}
PROPERTY FINAL Full : BOOL
GET
Full := _StaticCapacity <> 0 AND_THEN _Length >= _StaticCapacity;
END_GET
END_PROPERTY

(*!
<summary>Borrows the entry at a current storage position.</summary>
<description>
The index must be within Length and is not a sorted rank; otherwise an exception is raised. The returned
descriptor reference and payload remain collection-owned or borrowed from their original owner. Do not mutate
the descriptor or dispose of its payload through this view. Mutation or destruction may invalidate the
reference. Descendants cannot override this storage operation; capacity, indexing and disposal remain governed
by this collection implementation.
</description>
*)
METHOD FINAL GetByIndex : REFERENCE TO TOF_Core.GENERIC_VALUE
VAR_INPUT
	index : DINT;
END_VAR
IF index < 0 OR_ELSE index >= _Length THEN
	TOF_Core.Exceptions.ThrowArgumentOutOfRange(
		sourceNamespaceName := NamespaceName,
		sourceClassName := ClassName,
		sourcePOUName := __POUNAME(),
		sourcePosition := __POSITION(),
		argumentName := 'index',
		argumentValue := index
	);
END_IF

GetByIndex REF= _Array[index];
END_METHOD

(*!
<summary>Returns the matching entry position, or a negative value when absent.</summary>
<description>
The query is borrowed by default. Explicit release requests disposal of owned query storage after lookup
completes, including a missing result. Requested release is attempted after both successful lookup and lookup
failure. Before cleanup, the original framework exception is retained and a borrowed static system exception
is cloned to preserve its code, catch point and timestamps across cleanup callbacks. The captured exception is
then propagated through ExceptionManager.Throw in the current cyclic task; native errors use the framework
SystemException representation. If capturing the system exception fails with terminal OOM, query cleanup is
still attempted and terminal OOM takes precedence. Terminal allocation state is never cleared. Release is best
effort and does not prove successful deallocation. Cleanup callbacks must not reenter collection mutation.
Release resets only the local descriptor copy; the caller must have disposal rights and must not reuse or
release owning aliases afterwards. Borrowed payload is not freed. The position is a current storage slot with
no sorted-rank guarantee; mutation may invalidate it. Descendants cannot override this storage operation;
capacity, indexing and disposal remain governed by this collection implementation.
</description>
*)
METHOD FINAL GetGenericValuePosition : DINT
VAR_INPUT
	value : TOF_Core.GENERIC_VALUE;
	releaseValue : BOOL := FALSE;
END_VAR
VAR
	exceptionCode : __SYSTEM.ExceptionCode;
	caughtException : TOF_Core.IException;
END_VAR
__TRY
	IF NOT FindIndex(value := value, supposedIndex => GetGenericValuePosition) THEN
		GetGenericValuePosition := -1;
	END_IF
__CATCH(exceptionCode)
	caughtException := TOF_Core.ExceptionManager.GetLastException(
		exceptionCode := exceptionCode,
		catchPointNamespaceName := NamespaceName,
		catchPointPOUName := __POUNAME(),
		catchPointPosition := __POSITION()
	);
__ENDTRY

IF releaseValue THEN
	IF caughtException <> 0 AND_THEN NOT caughtException.IsDynamicInstance THEN
		__TRY
			TOF_Core.DynamicMemoryManager.RaiseIfAllocationFailed();
			__QUERYINTERFACE(caughtException.Clone(), caughtException);
		__CATCH(exceptionCode)
			value.Release();

			TOF_Core.ExceptionManager.ReThrowLastException(
				exceptionCode := exceptionCode,
				catchPointNamespaceName := NamespaceName,
				catchPointPOUName := __POUNAME(),
				catchPointPosition := __POSITION()
			);
		__ENDTRY
	END_IF

	value.Release();
END_IF

IF caughtException <> 0 THEN
	TOF_Core.ExceptionManager.Throw(exception := caughtException);
END_IF
END_METHOD

(*!
<summary>Returns the matching storage position, or a negative value when absent.</summary>
<description>
The raw ANY argument is borrowed without cloning or ownership transfer. isObject = TRUE requires a live Object
function-block instance, not a pointer or interface variable. FALSE uses ordinary runtime type mapping. The
caller keeps the query storage alive for the call. The position is a current storage slot with no sorted-rank
guarantee; mutation may invalidate it. Descendants cannot override this storage operation; capacity, indexing
and disposal remain governed by this collection implementation.
</description>
*)
//!<param name="isObject">Explicitly interprets the raw argument as a live Object instance.</param>
METHOD FINAL GetValuePosition : DINT
VAR_INPUT
	value : ANY;
	isObject : BOOL := FALSE;
END_VAR
VAR
	genericValue : TOF_Core.GENERIC_VALUE;
END_VAR

genericValue := TOF_Core.GenericValueFactory.FromAnyType(
		value := value,
		isObject := isObject,
		memoryManagementBehavior := TOF_Core.GENERIC_MEMORY_MANAGEMENT_BEHAVIOR.STORE_ORIGINAL_REFERENCE_AND_NOT_OWNS_MEMORY
	);

IF NOT FindIndex(value := genericValue, supposedIndex => GetValuePosition) THEN
	GetValuePosition := -1;
END_IF
END_METHOD

(*!
<summary>Reports the number of stored entries.</summary>
<description>
Units are bytes for ByteList and entries for other collections. Existing positions range from zero through
Length minus one.
</description>
*)
{attribute 'monitoring' := 'call'}
PROPERTY FINAL Length : TOF_Core.DINT_LENGTH
GET
Length := _Length;
END_GET
END_PROPERTY

(*!
<summary>Provides the library namespace for diagnostics.</summary>
<description>
Borrowed read-only reference to compiler-initialized metadata; no ownership transfer.
</description>
*)
{attribute 'monitoring' := 'call'}
PROPERTY NamespaceName : REFERENCE TO STRING
GET
NamespaceName REF= CurrentNamespace.Name;
END_GET
END_PROPERTY

(*!
<summary>Rebuilds bucket chains from cached hashes after entry relocation or capacity changes.</summary>
<description>
Requires bound index storage for positive capacity and valid hashes for every live entry. Does not allocate,
access payload or invoke callbacks. This only rebuilds links; it does not recompute hashes after
equality-relevant payload or address changes.
</description>
*)
METHOD PRIVATE rebuildIndex
VAR
	index : DINT;
	bucketIndex : DINT;
END_VAR
IF Capacity = TOF_Core.SignedInt32.ZERO THEN
	RETURN;
END_IF

Tc2_System.MEMSET(destAddr := _Buckets, fillByte := 0, n := TO_UDINT(XSIZEOF(DINT) * TO_ULINT(Capacity)));

FOR index := 0 TO _Length - 1 DO
	bucketIndex := TO_DINT(_Hashes[index] MOD TO_UDINT(Capacity));
	_NextIndices[index] := _Buckets[bucketIndex];
	_Buckets[bucketIndex] := index + 1;
END_FOR
END_METHOD

(*!
<summary>Removes the entry at a current storage position.</summary>
<description>
The index must be within Length and is not a sorted rank. Entries after the removed slot are compacted and
bucket links rebuilt from cached hashes before owned payload cleanup. Index compaction and rebuilding invoke
no equality/hash callbacks and allocate no storage. Invalid indices raise an exception. Positions and borrowed
entry references may be invalidated. Payload disposal is best effort through GENERIC_VALUE.Release.
Descendants cannot override this storage operation; capacity, indexing and disposal remain governed by this
collection implementation.
</description>
*)
METHOD FINAL RemoveAt : IUniqueDataSet
VAR_INPUT
	index : DINT;
END_VAR
VAR
	removedValue : TOF_Core.GENERIC_VALUE;
END_VAR
IF index < TOF_Core.SignedInt32.ZERO OR_ELSE index >= _Length THEN
	TOF_Core.Exceptions.ThrowArgumentOutOfRange(
		sourceNamespaceName := NamespaceName,
		sourceClassName := ClassName,
		sourcePOUName := __POUNAME(),
		sourcePosition := __POSITION(),
		argumentName := 'index',
		argumentValue := index
	);
END_IF

RemoveAt := THIS^;
removedValue := _Array[index];

IF index < _Length - 1 THEN
	Tc2_System.MEMMOVE(
		destAddr := ADR(_Array[index]),
		srcAddr := ADR(_Array[index + 1]),
		n := TO_UDINT(XSIZEOF(TOF_Core.GENERIC_VALUE) * TO_ULINT(_Length - index - 1))
	);
	Tc2_System.MEMMOVE(
		destAddr := ADR(_Hashes[index]),
		srcAddr := ADR(_Hashes[index + 1]),
		n := TO_UDINT(XSIZEOF(UDINT) * TO_ULINT(_Length - index - 1))
	);
END_IF

_Array[_Length - 1].Reset();
_Length := _Length - 1;
rebuildIndex();

removedValue.Release();
END_METHOD

(*!
<summary>Reports the size of this function-block instance.</summary>
<description>
Measured in bytes; includes inline storage but excludes separately allocated buffers, payload and enumerators.
</description>
*)
{attribute 'monitoring' := 'call'}
PROPERTY SelfSize : ULINT
GET
SelfSize := XSIZEOF(THIS^);
END_GET
END_PROPERTY

(*!
<summary>Copies a value and stores it through SetGeneric.</summary>
<description>
Borrows the original during the call. isObject = TRUE requires a live Object FB instance implementing
ICloneable; other data is copied as bytes without recursively cloning references. A prepared copy is released
if insertion fails before acceptance; exceptions propagate. Engine-managed exception objects are unsupported.
Any index output is meaningful only on success. Descendants cannot override this storage operation; capacity,
indexing and disposal remain governed by this collection implementation.
The original failure is captured before cleanup so nested cleanup handling cannot replace its payload.
A static native wrapper is cloned before cleanup; failure to capture still attempts prepared-copy disposal.
Terminal allocation failure takes precedence and no exception clone is allocated after its latch is set.
</description>
*)
METHOD FINAL SetCopy : IUniqueDataSet
VAR_INPUT
	value : ANY;
	isObject : BOOL := FALSE;
END_VAR
VAR_OUTPUT
	index : DINT;
END_VAR
VAR
	exceptionCode : __SYSTEM.ExceptionCode;
	caughtException : TOF_Core.IException;
	genericValue : TOF_Core.GENERIC_VALUE;
END_VAR

genericValue := TOF_Core.GenericValueFactory.FromAnyType(
		value := value,
		isObject := isObject,
		memoryManagementBehavior := TOF_Core.GENERIC_MEMORY_MANAGEMENT_BEHAVIOR.CLONE_ORIGINAL_VALUE_AND_OWNS_MEMORY
	);

__TRY
	SetCopy := SetGeneric(value := genericValue, index => index);
__CATCH(exceptionCode)
	caughtException := TOF_Core.ExceptionManager.GetLastException(
		exceptionCode := exceptionCode,
		catchPointNamespaceName := NamespaceName,
		catchPointPOUName := __POUNAME(),
		catchPointPosition := __POSITION()
	);
__ENDTRY

IF caughtException <> 0 THEN
	__TRY
		TOF_Core.DynamicMemoryManager.RaiseIfAllocationFailed();

		IF NOT caughtException.IsDynamicInstance THEN
			__QUERYINTERFACE(caughtException.Clone(), caughtException);
		END_IF
	__CATCH(exceptionCode)
		genericValue.Release();

		TOF_Core.ExceptionManager.ReThrowLastException(
			exceptionCode := exceptionCode,
			catchPointNamespaceName := NamespaceName,
			catchPointPOUName := __POUNAME(),
			catchPointPosition := __POSITION()
		);
	__ENDTRY

	genericValue.Release();

	TOF_Core.ExceptionManager.Throw(exception := caughtException);
END_IF
END_METHOD

(*!
<summary>Inserts a value or replaces the matching entry with the incoming descriptor.</summary>
<description>
Uses the lifetime equality/hash strategy, with no ordering guarantee. Empty descriptors are permitted unless
rejected by a validator. A successful call accepts incoming owned storage; borrowed payload must remain alive
while stored. Validation, lookup and growth precede acceptance; failure before acceptance leaves ownership
with the caller. A displaced owned allocation is released after replacement. Reusing the same allocation does
not release it and preserves existing ownership or accepts incoming ownership, without implicitly returning
ownership to the caller. Caller-side descriptor copies are not reset; transferred owning aliases must not be
released or reused as owners. Aliases must have compatible disposal semantics; overlapping owned ranges and
ownership already held by another entry or owner are not supported. Callbacks must not mutate or reenter this
collection. Cleanup through GENERIC_VALUE.Release is best effort and does not guarantee deallocation. The
index output is valid only on success. Descendants cannot override this storage operation; capacity, indexing
and disposal remain governed by this collection implementation.
</description>
*)
//!<param name="value">Incoming descriptor; owned storage is transferred on success.</param>
METHOD FINAL SetGeneric : IUniqueDataSet
VAR_INPUT
	value : TOF_Core.GENERIC_VALUE;
END_VAR
VAR_OUTPUT
	index : DINT;
END_VAR
VAR

	supposedIndex : DINT;
	hashCode : UDINT;
	bucketIndex : DINT;

	displacedValue : TOF_Core.GENERIC_VALUE;
END_VAR
IF _ValueValidator <> 0 THEN
	_ValueValidator.Validate(validatedObjectName := GetName(), valueToValidate := value);
END_IF

SetGeneric := THIS^;

IF FindIndex(value := value, supposedIndex => supposedIndex, hashCode => hashCode) THEN
	displacedValue := _Array[supposedIndex];

	IF displacedValue.Address = value.Address THEN
		IF displacedValue.IsMemoryOwner AND_THEN NOT value.IsMemoryOwner THEN
			value := TOF_Core.GenericValueFactory.FromParts(
				genericTypeClass := value.TypeClass,
				address := value.Address,
				size := value.Size,
				memoryManagementBehavior := TOF_Core.GENERIC_MEMORY_MANAGEMENT_BEHAVIOR.STORE_ORIGINAL_REFERENCE_AND_OWNS_MEMORY
			);
		END_IF

		displacedValue.Reset();
	END_IF
ELSE
	IF _Length >= Capacity THEN
		IF Dynamic THEN
			AllocateMemory(elementCount := DefaultDynamicAllocationElementCount);
		ELSE
			TOF_Core.Exceptions.ThrowStaticCollectionFull(
				sourceNamespaceName := NamespaceName,
				sourceClassName := ClassName,
				sourcePOUName := __POUNAME(),
				sourcePosition := __POSITION(),
				collectionName := GetName(),
				capacity := TO_UDINT(Capacity)
			);
		END_IF
	END_IF
END_IF

_Array[supposedIndex] := value;

IF supposedIndex = _Length THEN
	_Hashes[supposedIndex] := hashCode;
	bucketIndex := TO_DINT(hashCode MOD TO_UDINT(Capacity));
	_NextIndices[supposedIndex] := _Buckets[bucketIndex];
	_Buckets[bucketIndex] := supposedIndex + 1;
	_Length := _Length + 1;
END_IF

displacedValue.Release();

index := supposedIndex;
END_METHOD

(*!
<summary>Attempts to remove a matching entry.</summary>
<description>
Returns the collection for chaining. removed is TRUE only after the matching entry has been removed; FALSE
means no completed removal was reported. Removal is not transactional and does not prove successful
destruction of an owned payload. Catches exceptions without propagating them or clearing terminal allocation
state. Partial changes are not rolled back. The raw ANY argument is borrowed without cloning or ownership
transfer. isObject = TRUE requires a live Object function-block instance, not a pointer or interface variable.
FALSE uses ordinary runtime type mapping. The caller keeps the query storage alive for the call. Descendants
cannot override this storage operation; capacity, indexing and disposal remain governed by this collection
implementation.
After nested calls and requested cleanup, a fatal allocation state forces the reported outcome to failure.
This does not roll back completed removal or reset the application-wide fatal latch.
</description>
*)
//!<param name="isObject">Explicitly interprets the raw argument as a live Object instance.</param>
METHOD FINAL TryRemove : IUniqueDataSet
VAR_INPUT
	value : ANY;
	isObject : BOOL := FALSE;
END_VAR
VAR_OUTPUT
	removed : BOOL;
END_VAR
VAR
	genericValue : TOF_Core.GENERIC_VALUE;
	index : DINT;
END_VAR
TryRemove := THIS^;
removed := FALSE;

__TRY
	genericValue := TOF_Core.GenericValueFactory.FromAnyType(
		value := value,
		isObject := isObject,
		memoryManagementBehavior := TOF_Core.GENERIC_MEMORY_MANAGEMENT_BEHAVIOR.STORE_ORIGINAL_REFERENCE_AND_NOT_OWNS_MEMORY
	);

	IF FindIndex(value := genericValue, supposedIndex => index) THEN
		RemoveAt(index := index);
		removed := TRUE;
	END_IF
__CATCH
	removed := FALSE;
__ENDTRY

IF TOF_Core.DynamicMemoryManager.HasAllocationFailed THEN
	removed := FALSE;
END_IF
END_METHOD

(*!
<summary>Attempts to remove a matching entry.</summary>
<description>
Returns the collection for chaining. removed is TRUE only after the matching entry has been removed; FALSE
means no completed removal was reported. Removal is not transactional and does not prove successful
destruction of an owned payload. Catches exceptions without propagating them or clearing terminal allocation
state. Partial changes are not rolled back. The query is borrowed by default. When releaseValue is explicitly
TRUE, attempts to release the supplied generic argument after lookup/removal even on failure. The caller must
have disposal rights and must not reuse aliases of an owned argument after release. Descendants cannot
override this storage operation; capacity, indexing and disposal remain governed by this collection
implementation.
After nested calls and requested cleanup, a fatal allocation state forces the reported outcome to failure.
This does not roll back completed removal or reset the application-wide fatal latch.
</description>
*)
METHOD FINAL TryRemoveGeneric : IUniqueDataSet
VAR_INPUT
	value : TOF_Core.GENERIC_VALUE;
	releaseValue : BOOL := FALSE;
END_VAR
VAR_OUTPUT
	removed : BOOL;
END_VAR
VAR
	index : DINT;
END_VAR
TryRemoveGeneric := THIS^;
removed := FALSE;

__TRY
	IF FindIndex(value := value, supposedIndex => index) THEN
		RemoveAt(index := index);
		removed := TRUE;
	END_IF
__CATCH
	removed := FALSE;
__ENDTRY

IF releaseValue THEN
	__TRY
		value.Release();
	__CATCH
		removed := FALSE;
	__ENDTRY
END_IF

IF TOF_Core.DynamicMemoryManager.HasAllocationFailed THEN
	removed := FALSE;
END_IF
END_METHOD

(*!
<summary>Exposes the configured value validator.</summary>
<description>
Borrowed optional reference fixed at initialization. Zero means no validator. The collection does not own or
release it.
</description>
*)
{attribute 'monitoring' := 'call'}
PROPERTY FINAL ValueValidator : TOF_Core.IGenericValueValidator
GET
ValueValidator := _ValueValidator;
END_GET
END_PROPERTY

END_FUNCTION_BLOCK

// ---- UniqueDataSet/UniqueDataSetEnumerator.TcPOU
(*
SPDX-FileCopyrightText: © 2026 Oleksandr Tiutyk <trofimich@gmail.com>
SPDX-License-Identifier: MIT
License: https://opensource.org/license/mit
*)

(*!
<summary>Enumerates the current storage slots of a UniqueDataSet.</summary>
<description>
The source is borrowed and must outlive the cursor. Enumeration has no guaranteed ordering. Do not mutate the
source during traversal. Current is a borrowed view and must not be released or modified as an owning
descriptor; it is invalidated by cursor advancement/reset or source mutation. The caller owns and explicitly
releases a dynamically created cursor. MoveNext stops advancing at the end position of an unchanged source;
repeated exhausted calls return FALSE until Reset.
A null constructor source is diagnosed by traversal/current access, never by FB_init.
</description>
*)

{attribute 'no_explicit_call' := 'do not call this function block directly'}
{attribute 'enable_dynamic_creation'}
FUNCTION_BLOCK UniqueDataSetEnumerator EXTENDS TOF_Core.Object IMPLEMENTS TOF_Core.IEnumerator
VAR_STAT
	//! <summary>Class name shared by all instances of this function block.</summary>
	{attribute 'hide'} 
	_ClassName : STRING := __POUNAME();
END_VAR
VAR
	{attribute 'hide'} 
	_UniqueSet : IReadOnlyUniqueDataSet;
	{attribute 'hide'} 
	_CurrentIndex : DINT := -1;
	
	{attribute 'hide'} 
	_GenericValue : TOF_Core.GENERIC_VALUE;
END_VAR

(*!
<summary>Borrows the concrete cursor class name without transferring storage ownership.</summary>
*)
{attribute 'monitoring' := 'call'}
PROPERTY ClassName : REFERENCE TO STRING
GET
ClassName REF= _ClassName;
END_GET
END_PROPERTY

(*!
<summary>Exposes a read-only borrowed view of the current entry.</summary>
<description>
Reading Current before the first successful MoveNext, after Reset or after exhaustion yields an empty
descriptor. Otherwise payload is borrowed, with no disposal rights. Do not modify or release the descriptor.
The view may change on subsequent property access, cursor movement or source mutation.
Missing source raises DataMemberNotSpecifiedException before source access or cursor advancement.
</description>
*)
{attribute 'monitoring' := 'call'}
PROPERTY FINAL Current : REFERENCE TO TOF_Core.GENERIC_VALUE
GET
requireSource();

IF _CurrentIndex >= 0 AND_THEN _CurrentIndex < _UniqueSet.Length THEN
	_GenericValue := _UniqueSet.GetByIndex(index := _CurrentIndex); 
ELSE
	_GenericValue.Reset();	
END_IF 

Current REF= _GenericValue;
END_GET
END_PROPERTY

(*!
<summary>Binds the borrowed source for enumeration.</summary>
<description>
The source must be non-null and outlive the cursor. Only the reference is assigned; no allocation, callbacks
or throwing validation are performed. A null source remains invalid configuration and is reported by
MoveNext or current-value access without throwing from initialization.
</description>
*)
METHOD FB_init : BOOL
VAR_INPUT
	bInitRetains : BOOL; // TRUE: the retain variables are initialized (reset warm / reset cold)
	bInCopyCode : BOOL;  // TRUE: the instance will be copied to the copy code afterward (online change)
	uniqueSet : IReadOnlyUniqueDataSet;
END_VAR
_UniqueSet := uniqueSet;
END_METHOD

(*!
<summary>Advances the cursor to the next source position.</summary>
<description>
The source must be live, non-null and structurally unchanged during traversal. TRUE identifies a current
entry. The index advances only while below source Length and stops at the end position. Repeated exhausted
calls return FALSE without incrementing the index; reading Current yields an empty descriptor. Reset allows
traversal from the beginning again. No snapshot or mutation detection is provided. Descendants cannot override
this cursor operation; advancement, reset and borrowed current views use the same cursor state.
Missing source raises DataMemberNotSpecifiedException before source access or cursor advancement.
</description>
*)
{attribute "object_name" := "MoveNext"}
METHOD FINAL MoveNext : BOOL
requireSource();

IF _CurrentIndex < _UniqueSet.Length THEN
	_CurrentIndex := _CurrentIndex + 1;
END_IF

MoveNext := _CurrentIndex < _UniqueSet.Length;
END_METHOD

(*!
<summary>Provides the library namespace for diagnostics.</summary>
<description>
Borrowed read-only reference to compiler-initialized metadata; no ownership transfer.
</description>
*)
{attribute 'monitoring' := 'call'}
PROPERTY NamespaceName : REFERENCE TO STRING
GET
NamespaceName REF= CurrentNamespace.Name;
END_GET
END_PROPERTY

(*!
<summary>Places the cursor before the first source entry.</summary>
<description>
The next MoveNext starts at zero. Does not modify the source or release payload; reading Current now yields an
empty descriptor. Descendants cannot override this cursor operation; advancement, reset and borrowed current
views use the same cursor state.
</description>
*)
{attribute "object_name" := "Reset"}
METHOD FINAL Reset
_CurrentIndex := -1;
END_METHOD

(*!
<summary>Reports the size of this function-block instance.</summary>
<description>
Measured in bytes; includes inline storage but excludes separately allocated buffers, payload and enumerators.
</description>
*)
{attribute 'monitoring' := 'call'}
PROPERTY SelfSize : ULINT
GET
SelfSize := XSIZEOF(THIS^);
END_GET
END_PROPERTY

(*!
<summary>Requires the configured source before traversal or current-value access.</summary>
<description>
A missing mandatory source is configuration failure, not an empty collection. Raises a framework diagnostic
outside lifecycle methods and before mutation; it does not validate arbitrary pointer lifetime.
</description>
*)
METHOD PRIVATE requireSource
IF _UniqueSet = 0 THEN
	TOF_Core.Exceptions.ThrowDataMemberNotSpecified(
		sourceNamespaceName := NamespaceName,
		sourceClassName := ClassName,
		sourcePOUName := __POUNAME(),
		sourcePosition := __POSITION(),
		dataMemberName := 'uniqueSet'
	);
END_IF
END_METHOD

END_FUNCTION_BLOCK
